TYPE ST_KBUS_AnalogueDataOut :
STRUCT
	nCtrl	: BYTE;
	nData	: INT;
END_STRUCT
END_TYPE

(* stored: Version 1.1.0.1
   DUT ST_KBUS_AnalogueDataOut: Id {e0c114e5-87e1-42b6-be7c-0adc44cc9136} *)
